// TIA Portal V17 export
// export: Created 2024-08-29T18:23:45.096152Z, ExportSetting WithDefaults, DisplayName Totally Integrated Automation Portal, DisplayVersion V17 Update 7, DisplayName TIA Portal Openness, DisplayVersion V17 Update 7, DisplayName TIA Portal Version Control Interface, DisplayVersion V17, DisplayName SINAMICS Startdrive Advanced, DisplayVersion V17 SP2, DisplayName SINAMICS Startdrive G110M, G120, G120C, G120D, G120P, G115D, DisplayVersion V17 SP2, DisplayName SINAMICS Startdrive G130, G150, S120, S150, SINAMICS MV, S210, DisplayVersion V17 SP2, DisplayName STEP 7 Professional, DisplayVersion V17 Update 7, DisplayName STEP 7 Safety, DisplayVersion V17 Update 6, DisplayName WinCC Advanced / Unified PC, DisplayVersion V17 Update 7
DATA_BLOCK "DB_ControlPrinter"   // DB2500
VERSION : 0.1
// stored: AutoNumber false, DBAccessibleFromOPCUA true, DBAccessibleFromWebserver true, InstanceOfName FB_ControlPrinter, InstanceOfType FB
"FB_ControlPrinter"
   // VAR_INPUT
   //    printNewLabel : Bool := FALSE;
   //    printLastLabel : Bool := FALSE;
   //    printBlackLabel : Bool := FALSE;
   //    resetLabelCounter : Bool := FALSE;
   //    resetErrors : Bool := FALSE;
   //    typeOfLabel : Int := 1;
   //    optionAutoResetCounter : Int := 0;
   //    REF_TO_PRINT_PLANT_NUMER_3DIGIT : String[10] := 'YRN';
   //    NFP : String[30] := '';
   //    Traceability : Bool := FALSE;
   //    line : String[1] := '2';
   //    reference : "udt_referenceMainInfo";
   // END_VAR
   // VAR_OUTPUT
   //    printDone : Bool := FALSE;
   //    printBusy : Bool := FALSE;
   //    printError : Bool := FALSE;
   //    printerStatus : Word := 16#7004;
   // END_VAR
   // VAR
   //    tramToSendToPrinter : Array[0..6000] of Char;
   //    seqDataPreparation : Int := 0;
   //    tramToPrepareToSend { S7_SetPoint := 'True'} : Array[1..20] of String;
   //    savePrintNewLabel : Bool := FALSE;
   // END_VAR
   // VAR RETAIN
   //    "counter" : Int := 50;
   //    DBcomToPrinter : TCON_IP_v4;
   // END_VAR
   // VAR
   //    tSendC { S7_SetPoint := 'True'} : TSEND_C;
   // END_VAR
BEGIN
   reference.id := 0;
   reference.description := 'xxxxx';
   reference.partNumber := '2799821X';
   reference.rev := '05';
   reference.customerNumber := '13543982';
   reference.vpps := '4270100000000L';
   reference.locationCode := '7';
   reference.dataIdentifier := '888';
   reference.duns := '812785841';
   tramToSendToPrinter[0] := '^';
   tramToSendToPrinter[1] := 'X';
   tramToSendToPrinter[2] := 'A';
   tramToSendToPrinter[3] := '^';
   tramToSendToPrinter[4] := 'P';
   tramToSendToPrinter[5] := 'W';
   tramToSendToPrinter[6] := '3';
   tramToSendToPrinter[7] := '7';
   tramToSendToPrinter[8] := '8';
   tramToSendToPrinter[9] := '^';
   tramToSendToPrinter[10] := 'B';
   tramToSendToPrinter[11] := 'Y';
   tramToSendToPrinter[12] := '1';
   tramToSendToPrinter[13] := '2';
   tramToSendToPrinter[14] := '6';
   tramToSendToPrinter[15] := ',';
   tramToSendToPrinter[16] := '1';
   tramToSendToPrinter[17] := '2';
   tramToSendToPrinter[18] := '6';
   tramToSendToPrinter[19] := '^';
   tramToSendToPrinter[20] := 'F';
   tramToSendToPrinter[21] := 'T';
   tramToSendToPrinter[22] := '1';
   tramToSendToPrinter[23] := '6';
   tramToSendToPrinter[24] := '9';
   tramToSendToPrinter[25] := ',';
   tramToSendToPrinter[26] := '1';
   tramToSendToPrinter[27] := '7';
   tramToSendToPrinter[28] := '5';
   tramToSendToPrinter[29] := '^';
   tramToSendToPrinter[30] := 'B';
   tramToSendToPrinter[31] := 'X';
   tramToSendToPrinter[32] := 'N';
   tramToSendToPrinter[33] := ',';
   tramToSendToPrinter[34] := '7';
   tramToSendToPrinter[35] := ',';
   tramToSendToPrinter[36] := '2';
   tramToSendToPrinter[37..38] := '0';
   tramToSendToPrinter[39] := ',';
   tramToSendToPrinter[40] := '0';
   tramToSendToPrinter[41] := ',';
   tramToSendToPrinter[42] := '0';
   tramToSendToPrinter[43] := ',';
   tramToSendToPrinter[44] := '1';
   tramToSendToPrinter[45] := ',';
   tramToSendToPrinter[46] := '~';
   tramToSendToPrinter[47] := '^';
   tramToSendToPrinter[48] := 'F';
   tramToSendToPrinter[49] := 'H';
   tramToSendToPrinter[50] := '\';
   tramToSendToPrinter[51] := '^';
   tramToSendToPrinter[52] := 'F';
   tramToSendToPrinter[53] := 'D';
   tramToSendToPrinter[54] := '2';
   tramToSendToPrinter[55] := 'P';
   tramToSendToPrinter[56] := '0';
   tramToSendToPrinter[57] := '5';
   tramToSendToPrinter[58] := '0';
   tramToSendToPrinter[59] := 'H';
   tramToSendToPrinter[60] := '2';
   tramToSendToPrinter[61] := '1';
   tramToSendToPrinter[62] := '5';
   tramToSendToPrinter[63] := '4';
   tramToSendToPrinter[64..65] := '1';
   tramToSendToPrinter[66] := '8';
   tramToSendToPrinter[67] := '0';
   tramToSendToPrinter[68..69] := '9';
   tramToSendToPrinter[70] := 'R';
   tramToSendToPrinter[71] := '0';
   tramToSendToPrinter[72] := '1';
   tramToSendToPrinter[73] := 'Y';
   tramToSendToPrinter[74] := 'R';
   tramToSendToPrinter[75] := 'N';
   tramToSendToPrinter[76] := '2';
   tramToSendToPrinter[77] := '4';
   tramToSendToPrinter[78] := '^';
   tramToSendToPrinter[79] := 'F';
   tramToSendToPrinter[80] := 'S';
   tramToSendToPrinter[81] := '^';
   tramToSendToPrinter[82] := 'F';
   tramToSendToPrinter[83] := 'T';
   tramToSendToPrinter[84] := '2';
   tramToSendToPrinter[85] := '5';
   tramToSendToPrinter[86] := ',';
   tramToSendToPrinter[87] := '1';
   tramToSendToPrinter[88] := '6';
   tramToSendToPrinter[89] := '2';
   tramToSendToPrinter[90] := '^';
   tramToSendToPrinter[91] := 'A';
   tramToSendToPrinter[92] := '0';
   tramToSendToPrinter[93] := 'N';
   tramToSendToPrinter[94] := ',';
   tramToSendToPrinter[95] := '2';
   tramToSendToPrinter[96] := '9';
   tramToSendToPrinter[97] := ',';
   tramToSendToPrinter[98] := '2';
   tramToSendToPrinter[99] := '8';
   tramToSendToPrinter[100] := '^';
   tramToSendToPrinter[101] := 'F';
   tramToSendToPrinter[102] := 'H';
   tramToSendToPrinter[103] := '\';
   tramToSendToPrinter[104] := '^';
   tramToSendToPrinter[105] := 'F';
   tramToSendToPrinter[106] := 'D';
   tramToSendToPrinter[107] := '4';
   tramToSendToPrinter[108..109] := '1';
   tramToSendToPrinter[110] := '8';
   tramToSendToPrinter[111] := '0';
   tramToSendToPrinter[112..113] := '9';
   tramToSendToPrinter[114] := '^';
   tramToSendToPrinter[115] := 'F';
   tramToSendToPrinter[116] := 'S';
   tramToSendToPrinter[117] := '^';
   tramToSendToPrinter[118] := 'F';
   tramToSendToPrinter[119] := 'T';
   tramToSendToPrinter[120] := '2';
   tramToSendToPrinter[121] := '5';
   tramToSendToPrinter[122] := ',';
   tramToSendToPrinter[123] := '1';
   tramToSendToPrinter[124] := '2';
   tramToSendToPrinter[125] := '4';
   tramToSendToPrinter[126] := '^';
   tramToSendToPrinter[127] := 'A';
   tramToSendToPrinter[128] := '0';
   tramToSendToPrinter[129] := 'N';
   tramToSendToPrinter[130] := ',';
   tramToSendToPrinter[131] := '2';
   tramToSendToPrinter[132] := '5';
   tramToSendToPrinter[133] := ',';
   tramToSendToPrinter[134] := '2';
   tramToSendToPrinter[135] := '4';
   tramToSendToPrinter[136] := '^';
   tramToSendToPrinter[137] := 'F';
   tramToSendToPrinter[138] := 'H';
   tramToSendToPrinter[139] := '\';
   tramToSendToPrinter[140] := '^';
   tramToSendToPrinter[141] := 'F';
   tramToSendToPrinter[142] := 'D';
   tramToSendToPrinter[143] := '0';
   tramToSendToPrinter[144] := '2';
   tramToSendToPrinter[145] := '/';
   tramToSendToPrinter[146] := '0';
   tramToSendToPrinter[147] := '8';
   tramToSendToPrinter[148] := '/';
   tramToSendToPrinter[149] := '2';
   tramToSendToPrinter[150] := '0';
   tramToSendToPrinter[151] := '2';
   tramToSendToPrinter[152] := '4';
   tramToSendToPrinter[153] := '^';
   tramToSendToPrinter[154] := 'F';
   tramToSendToPrinter[155] := 'S';
   tramToSendToPrinter[156] := '^';
   tramToSendToPrinter[157] := 'F';
   tramToSendToPrinter[158] := 'T';
   tramToSendToPrinter[159] := '2';
   tramToSendToPrinter[160] := '5';
   tramToSendToPrinter[161] := ',';
   tramToSendToPrinter[162] := '8';
   tramToSendToPrinter[163] := '7';
   tramToSendToPrinter[164] := '^';
   tramToSendToPrinter[165] := 'A';
   tramToSendToPrinter[166] := '0';
   tramToSendToPrinter[167] := 'N';
   tramToSendToPrinter[168] := ',';
   tramToSendToPrinter[169] := '2';
   tramToSendToPrinter[170] := '9';
   tramToSendToPrinter[171] := ',';
   tramToSendToPrinter[172] := '2';
   tramToSendToPrinter[173] := '8';
   tramToSendToPrinter[174] := '^';
   tramToSendToPrinter[175] := 'F';
   tramToSendToPrinter[176] := 'H';
   tramToSendToPrinter[177] := '\';
   tramToSendToPrinter[178] := '^';
   tramToSendToPrinter[179] := 'F';
   tramToSendToPrinter[180] := 'D';
   tramToSendToPrinter[181] := '0';
   tramToSendToPrinter[182] := '7';
   tramToSendToPrinter[183] := ':';
   tramToSendToPrinter[184] := '2';
   tramToSendToPrinter[185] := '7';
   tramToSendToPrinter[186] := ':';
   tramToSendToPrinter[187] := '3';
   tramToSendToPrinter[188] := '8';
   tramToSendToPrinter[189] := '^';
   tramToSendToPrinter[190] := 'F';
   tramToSendToPrinter[191] := 'S';
   tramToSendToPrinter[192] := '^';
   tramToSendToPrinter[193] := 'F';
   tramToSendToPrinter[194] := 'T';
   tramToSendToPrinter[195] := '2';
   tramToSendToPrinter[196] := '6';
   tramToSendToPrinter[197] := ',';
   tramToSendToPrinter[198..199] := '4';
   tramToSendToPrinter[200] := '^';
   tramToSendToPrinter[201] := 'A';
   tramToSendToPrinter[202] := '0';
   tramToSendToPrinter[203] := 'N';
   tramToSendToPrinter[204] := ',';
   tramToSendToPrinter[205] := '2';
   tramToSendToPrinter[206] := '9';
   tramToSendToPrinter[207] := ',';
   tramToSendToPrinter[208] := '2';
   tramToSendToPrinter[209] := '8';
   tramToSendToPrinter[210] := '^';
   tramToSendToPrinter[211] := 'F';
   tramToSendToPrinter[212] := 'H';
   tramToSendToPrinter[213] := '\';
   tramToSendToPrinter[214] := '^';
   tramToSendToPrinter[215] := 'F';
   tramToSendToPrinter[216] := 'D';
   tramToSendToPrinter[217] := 'H';
   tramToSendToPrinter[218] := '-';
   tramToSendToPrinter[219] := 'F';
   tramToSendToPrinter[220] := 'r';
   tramToSendToPrinter[221] := 'a';
   tramToSendToPrinter[222] := 'm';
   tramToSendToPrinter[223] := 'e';
   tramToSendToPrinter[224] := ' ';
   tramToSendToPrinter[225] := '4';
   tramToSendToPrinter[226] := 'W';
   tramToSendToPrinter[227] := ' ';
   tramToSendToPrinter[228] := 'R';
   tramToSendToPrinter[229] := 'H';
   tramToSendToPrinter[230] := '^';
   tramToSendToPrinter[231] := 'F';
   tramToSendToPrinter[232] := 'S';
   tramToSendToPrinter[233] := '^';
   tramToSendToPrinter[234] := 'F';
   tramToSendToPrinter[235] := 'T';
   tramToSendToPrinter[236] := '2';
   tramToSendToPrinter[237] := '5';
   tramToSendToPrinter[238] := ',';
   tramToSendToPrinter[239] := '1';
   tramToSendToPrinter[240] := '9';
   tramToSendToPrinter[241] := '6';
   tramToSendToPrinter[242] := '^';
   tramToSendToPrinter[243] := 'A';
   tramToSendToPrinter[244] := '0';
   tramToSendToPrinter[245] := 'N';
   tramToSendToPrinter[246] := ',';
   tramToSendToPrinter[247] := '2';
   tramToSendToPrinter[248] := '1';
   tramToSendToPrinter[249] := ',';
   tramToSendToPrinter[250] := '2';
   tramToSendToPrinter[251] := '1';
   tramToSendToPrinter[252] := '^';
   tramToSendToPrinter[253] := 'F';
   tramToSendToPrinter[254] := 'H';
   tramToSendToPrinter[255] := '\';
   tramToSendToPrinter[256] := '^';
   tramToSendToPrinter[257] := 'F';
   tramToSendToPrinter[258] := 'D';
   tramToSendToPrinter[259] := '2';
   tramToSendToPrinter[260] := 'P';
   tramToSendToPrinter[261] := '0';
   tramToSendToPrinter[262] := '5';
   tramToSendToPrinter[263] := '0';
   tramToSendToPrinter[264] := 'H';
   tramToSendToPrinter[265] := '2';
   tramToSendToPrinter[266] := '1';
   tramToSendToPrinter[267] := '5';
   tramToSendToPrinter[268] := '4';
   tramToSendToPrinter[269..270] := '1';
   tramToSendToPrinter[271] := '8';
   tramToSendToPrinter[272] := '0';
   tramToSendToPrinter[273..274] := '9';
   tramToSendToPrinter[275] := 'R';
   tramToSendToPrinter[276] := '0';
   tramToSendToPrinter[277] := '1';
   tramToSendToPrinter[278] := 'Y';
   tramToSendToPrinter[279] := 'R';
   tramToSendToPrinter[280] := 'N';
   tramToSendToPrinter[281] := '2';
   tramToSendToPrinter[282] := '4';
   tramToSendToPrinter[283] := '^';
   tramToSendToPrinter[284] := 'P';
   tramToSendToPrinter[285] := 'Q';
   tramToSendToPrinter[286] := '1';
   tramToSendToPrinter[287] := ',';
   tramToSendToPrinter[288] := '0';
   tramToSendToPrinter[289] := ',';
   tramToSendToPrinter[290] := '1';
   tramToSendToPrinter[291] := ',';
   tramToSendToPrinter[292] := 'Y';
   tramToSendToPrinter[293] := '^';
   tramToSendToPrinter[294] := 'X';
   tramToSendToPrinter[295] := 'Z';
   tramToSendToPrinter[296..6000] := ' ';
   tramToPrepareToSend[1] := '^XA^PW378';
   tramToPrepareToSend[2] := '^BY126,126^FT169,175^BXN,7,200,0,0,1,~^FH\^FD';
   tramToPrepareToSend[3] := '2P050H2154118099R01YRN24';
   tramToPrepareToSend[4] := '^FS^FT25,162^A0N,29,28^FH\^FD';
   tramToPrepareToSend[5] := '4118099';
   tramToPrepareToSend[6] := '^FS^FT25,124^A0N,25,24^FH\^FD';
   tramToPrepareToSend[7] := '02/08/2024';
   tramToPrepareToSend[8] := '^FS^FT25,87^A0N,29,28^FH\^FD';
   tramToPrepareToSend[9] := '07:27:38';
   tramToPrepareToSend[10] := '^FS^FT26,44^A0N,29,28^FH\^FD';
   tramToPrepareToSend[11] := 'H-Frame 4W RH';
   tramToPrepareToSend[12] := '^FS^FT25,196^A0N,21,21^FH\^FD';
   tramToPrepareToSend[13] := '2P050H2154118099R01YRN24';
   tramToPrepareToSend[14..19] := '';
   tramToPrepareToSend[20] := '^PQ1,0,1,Y^XZ';
   DBcomToPrinter.InterfaceId := 64;
   DBcomToPrinter.ID := 16#000A;
   DBcomToPrinter.ConnectionType := 16#0B;
   DBcomToPrinter.ActiveEstablished := TRUE;
   DBcomToPrinter.RemoteAddress.ADDR[1] := 16#C0;
   DBcomToPrinter.RemoteAddress.ADDR[2] := 16#A8;
   DBcomToPrinter.RemoteAddress.ADDR[3] := 16#01;
   DBcomToPrinter.RemoteAddress.ADDR[4] := 16#37;
   DBcomToPrinter.RemotePort := 6101;
   DBcomToPrinter.LocalPort := 0;
   tSendC.REQ := FALSE;
   tSendC.CONT := TRUE;
   tSendC.LEN := 0;
   tSendC.DONE := FALSE;
   tSendC.BUSY := FALSE;
   tSendC.ERROR := FALSE;
   tSendC.STATUS := 16#7004;
   tSendC.COM_RST := FALSE;
   tSendC.s_state := 3;
   tSendC.sb_udp := FALSE;
   tSendC.sb_b_REQ := FALSE;
   tSendC.tcon_80A3 := FALSE;
   tSendC.sw_ConID := 16#000A;
   tSendC.s_TCON.REQ := FALSE;
   tSendC.s_TCON.ID := 16#000A;
   tSendC.s_TCON.DONE := TRUE;
   tSendC.s_TCON.BUSY := FALSE;
   tSendC.s_TCON.ERROR := FALSE;
   tSendC.s_TCON.STATUS := 16#0000;
   tSendC.s_T_DIAG.REQ := FALSE;
   tSendC.s_T_DIAG.ID := 16#000A;
   tSendC.s_T_DIAG.DONE := TRUE;
   tSendC.s_T_DIAG.BUSY := FALSE;
   tSendC.s_T_DIAG.ERROR := FALSE;
   tSendC.s_T_DIAG.STATUS := 16#0000;
   tSendC.s_TDiag_Status.InterfaceId := 64;
   tSendC.s_TDiag_Status.ID := 16#000A;
   tSendC.s_TDiag_Status.ConnectionType := 16#0B;
   tSendC.s_TDiag_Status.ActiveEstablished := TRUE;
   tSendC.s_TDiag_Status.State := 16#04;
   tSendC.s_TDiag_Status.Kind := 16#03;
   tSendC.s_TDiag_Status.SentBytes := 0;
   tSendC.s_TDiag_Status.ReceivedBytes := 0;
   tSendC.s_TDISCON.REQ := FALSE;
   tSendC.s_TDISCON.ID := 16#000A;
   tSendC.s_TDISCON.DONE := FALSE;
   tSendC.s_TDISCON.BUSY := FALSE;
   tSendC.s_TDISCON.ERROR := FALSE;
   tSendC.s_TDISCON.STATUS := 16#7000;
   tSendC.s_TSEND.REQ := FALSE;
   tSendC.s_TSEND.ID := 16#000A;
   tSendC.s_TSEND.LEN := 0;
   tSendC.s_TSEND.DONE := TRUE;
   tSendC.s_TSEND.BUSY := FALSE;
   tSendC.s_TSEND.ERROR := FALSE;
   tSendC.s_TSEND.STATUS := 16#0000;
   tSendC.s_TUSEND.REQ := FALSE;
   tSendC.s_TUSEND.ID := 16#000A;
   tSendC.s_TUSEND.LEN := 0;
   tSendC.s_TUSEND.DONE := FALSE;
   tSendC.s_TUSEND.BUSY := FALSE;
   tSendC.s_TUSEND.ERROR := FALSE;
   tSendC.s_TUSEND.STATUS := 16#7000;
   tSendC.s_TRESET.REQ := FALSE;
   tSendC.s_TRESET.ID := 16#000A;
   tSendC.s_TRESET.DONE := FALSE;
   tSendC.s_TRESET.BUSY := FALSE;
   tSendC.s_TRESET.ERROR := FALSE;
   tSendC.s_TRESET.STATUS := 16#0000;
END_DATA_BLOCK
